# EPICS substitutions: GalilTestApp/Db/galil_rio_analog_ports.substitutions
# Description:
# adc/dac substitution file.
#
# This library is free software; you can redistribute it and/or
# modify it under the terms of the GNU Lesser General Public
# Licence as published by the Free Software Foundation; either
# version 2.1 of the Licence, or (at your option) any later version.
#
# This library is distributed in the hope that it will be useful,
# but WITHOUT ANY WARRANTY; without even the implied warranty of
# MERCHANTABILITY or FITNESS FOR A PARTICULAR PURPOSE.  See the GNU
# Lesser General Public Licence for more details.
#
# You should have received a copy of the GNU Lesser General Public
# Licence along with this library; if not, write to the Free Software
# Foundation, Inc., 51 Franklin St, Fifth Floor, Boston, MA 02110-1301 USA.
#
# Contact details:
# Mark Clift
# email: padmoz@tpg.com.au

# R    - Record Name
# ADDR - Hardware port to read
# PREC - Precision

file "$(GALIL)/GalilSup/Db/galil_analog_in.template"
{
   pattern { R,           ADDR,  SCAN,       PREC }

#RIO Ports numbered 0 to 7 on controller hardware
	   { "GalilAi0",  "0",   "I/O Intr", "3"  }
	   { "GalilAi1",  "1",   "I/O Intr", "3"  }
	   { "GalilAi2",  "2",   "I/O Intr", "3"  }
	   { "GalilAi3",  "3",   "I/O Intr", "3"  }
	   { "GalilAi4",  "4",   "I/O Intr", "3"  }
	   { "GalilAi5",  "5",   "I/O Intr", "3"  }
	   { "GalilAi6",  "6",   "I/O Intr", "3"  }
	   { "GalilAi7",  "7",   "I/O Intr", "3"  }
}

file "$(GALIL)/GalilSup/Db/galil_analog_out.template"
{
   pattern { R,           ADDR,  PREC,  LOPR,  HOPR }

#RIO Ports numbered 0 to 7 on controller hardware
	   { "GalilAo0",  "0",   "3",   "-10", "10" }
	   { "GalilAo1",  "1",   "3",   "-10", "10" }
	   { "GalilAo2",  "2",   "3",   "-10", "10" }
	   { "GalilAo3",  "3",   "3",   "-10", "10" }
	   { "GalilAo4",  "4",   "3",   "-10", "10" }
	   { "GalilAo5",  "5",   "3",   "-10", "10" }
	   { "GalilAo6",  "6",   "3",   "-10", "10" }
	   { "GalilAo7",  "7",   "3",   "-10", "10" }
}

# end
